TYPE ST_CFG_SingelSensor :
STRUCT
	Enable: BOOL; 
	Measurement_Value : INT;
END_STRUCT
END_TYPE

(* stored: Version 1.1.0.1, ProductVersion 3.1.4024.9
   DUT ST_CFG_SingelSensor: Id {33c91950-a7ff-4574-8b40-04f4b4cc65c1} *)
